(* IEC 61131-3 sources: AXOpen/src/messaging/ctrl/src/IxMessaging, 8 files *)

(* ---- eIxMessageCondition.st ---- *)
NAMESPACE ix.framework.core
    TYPE INTERNAL
        eIxMessageCondition : INT
        (
            Unconditional := 0,
            Active := 10,
            Inactive := 20
        );
    END_TYPE
END_NAMESPACE

(* ---- eIxMessageDigestMethod.st ---- *)
NAMESPACE ix.framework.core
    /// <summary>
    /// Message digest methods used to create fingerprint of a message.
    /// </summary>
    TYPE eIxMessageDigestMethod : INT
    (
        /// <summary>
        /// Fastest method with highest probability of colisions.
        /// </summary>
        CRC8 := 8,

        /// <summary>
        /// Moderate speed method with lower probability of colisions.
        /// </summary>
        CRC16 := 16,

        /// <summary>
        /// Slowest speed method with relatively low probability of colisions.
        /// </summary>
        CRC32 := 32,

        /// <summary>
        /// Messages are not digested the repeated messages won't be filtered out.
        /// Use this option on low performance devices.
        /// </summary>
        NONE := 32767
    );
    END_TYPE
END_NAMESPACE

(* ---- IxConstants.st ---- *)
NAMESPACE ix.framework.core
    TYPE PUBLIC
        IxIntConstants : INT
        (
            MAX_MESSAGE_TEXT_LENGHT := 160,
			MDS_MAX_INDEX := 10
        );
    END_TYPE
END_NAMESPACE

(* ---- IxMessage.st ---- *)
NAMESPACE ix.framework.messaging
    ///<summary>
    /// Complete message details including time stamp, message text, message category, identity of the message provider, context cycle in which the message was posted.
    ///</summary>
    TYPE IxMessage:
        STRUCT
            /// <summary>
            /// Time when the message was posted.
            /// </summary>
            {#ix-attr:[ReadOnly()]}
            TimeStamp : LDATE_AND_TIME;

            /// <summary>
            /// Text of the message.
            /// </summary>
            {#ix-attr:[ReadOnly()]}
            Text : STRING[IxIntConstants#MAX_MESSAGE_TEXT_LENGHT];

            /// <summary>
            /// Identity of the TcoObject that posted this message.
            /// </summary>
            {#ix-attr:[ReadOnly()]}
            Identity : ULINT;

            /// <summary>
            /// Message category of this message. See <see cref="TcoCore.eMessageCategory"/> for detailed informations.
            /// </summary>
            Category : eIxMessageCategory;

            /// <summary>
            /// Context cycle in which the message was posted.
            /// </summary>
            {#ix-attr:[ReadOnly()]}
            Cycle : ULINT;

            /// <summary>
            /// Count of messages of the object in the current cycle.
            /// </summary>
            {#ix-attr:[ReadOnly()]}
            PerCycleCount : USINT;

            /// <summary>
            /// Indicates that the message is expected to be dequeed from the buffer.
            /// </summary>
            ExpectDequeing : BOOL;

            /// <summary>
            /// Indicates that the message must be persisted in the alarm view until acknowledged.
            /// </summary>
            Pinned : BOOL;

            /// <summary>
            /// Stores message digest of this message text.
            /// </summary>
            MessageDigest : DWORD;

            // /// <summary>
            // /// Indicates that the message is active.
            // /// </summary>
            // IsActive : BOOL;
        END_STRUCT;
    END_TYPE
 END_NAMESPACE

(* ---- IxMessageDigest.st ---- *)
NAMESPACE ix.framework.messaging
    CLASS PUBLIC IxMessageDigest
        VAR PUBLIC
            Digest : DWORD;
            Cycle : ULINT;
            Count : ULINT;
            Category : eIxMessageCategory;
        END_VAR
    END_CLASS
END_NAMESPACE

(* ---- IxMessenger.st ---- *)
USING ix.framework.core;
USING System.Strings;
USING System.DateTime;
USING ix.framework.utils;
USING ix.framework.core;
USING ix.framework.messaging;

NAMESPACE ix.framework.messaging
	/// <summary>
	/// Provides mechanism for delivering static messages to the supervising applications (SCADA/HMI).
	/// 	<remarks>
	/// 		<note type="important">
	/// 			Each messenger has a single placeholder for the message; it stores the most important message from the last context cycle.
	/// 			If there are more messages in a single cycle for the same messenger then less important messages are discarded and replaced by
	/// 			the message with the category of higher severity.
	/// 		</note>
	/// 		<note type="important">
	/// 			Messenger can send the data to context logger. There is a maximum limit of 10 different messages per messenger in 2 consecutive context cycles.
	/// 			The messages that exceed this limit won't be logged when `OnEventRisen` logging is set.
	/// 		    Take this behaviour into account when designing your system.
	/// 		</note>
	/// 	</remarks>
	/// </summary>
    CLASS IxMessenger (*EXTENDS IxObject*) IMPLEMENTS IIxMessenger, IIxMessageProperties, IIxMessageTextBuilder, IIxMessageCategorize, IIxMessages
		VAR
			/// <summary>
			/// 	Most important message of this instance of messenger; stores the most important message from the last context cycle.
			/// 	If there are more messages in a single cycle for the same
			/// 	messenger then less important messages are discarded and replaced by the message with the category of higher severity.
			/// </summary>
			_mime : IxMessage;
			_Parent : IIxObject;
            {#ix-attr:[ReadOnly()]}
			_contextIdentity : ULINT;
			{#ix-attr:[CompilerOmits()]}
			_mds : ARRAY[0..IxIntConstants#MDS_MAX_INDEX] OF IxMessageDigest;
			{#ix-attr:[CompilerOmits()]}
			_condition : eIxMessageCondition;
			{#ix-attr:[CompilerOmits()]}
			_pinnable : BOOL;
		END_VAR

		VAR
			{#ix-attr:[CompilerOmits()]}
			tmpMessageText : STRING[IxIntConstants#MAX_MESSAGE_TEXT_LENGHT];
			{#ix-attr:[CompilerOmits()]}
			refStringBuilder : REF_TO StringBuilder;
		END_VAR
		VAR
			{#ix-attr:[CompilerOmits()]}
			_conflictingStringBuilder : StringBuilder;
		END_VAR

		/// <summary>
		/// Gets the Most Important Message of this messenger.
		/// </summary>
		METHOD PUBLIC GetMime : IxMessage
			GetMime := THIS._mime;
		END_METHOD

		/// <summary>
		/// Categorizes and creates the message as 'debug'.
		/// </summary>
		METHOD PUBLIC AsDebug : IIxMessageProperties
			AsDebug := THIS.Post(THIS.StringBuilder()^.AsString(), eIxMessageCategory#Debug);
		END_METHOD

		/// <summary>
		/// Categorizes and creates the message as 'error'.
		/// </summary>
		METHOD PUBLIC AsError : IIxMessageProperties
			AsError := THIS.Post(THIS.StringBuilder()^.AsString(), eIxMessageCategory#Error);
		END_METHOD

		/// <summary>
		/// Categorizes and creates the message as 'fatal'.
		/// </summary>
		METHOD PUBLIC AsFatal : IIxMessageProperties
			AsFatal := THIS.Post(THIS.StringBuilder()^.AsString(), eIxMessageCategory#Fatal);
		END_METHOD

		/// <summary>
		/// Categorizes and creates the message as 'information'.
		/// </summary>
		METHOD PUBLIC AsInfo : IIxMessageProperties
			AsInfo := THIS.Post(THIS.StringBuilder()^.AsString(), eIxMessageCategory#Info);
		END_METHOD

		/// <summary>
		/// Categorizes and creates the message as 'trace'.
		/// </summary>
		METHOD PUBLIC AsTrace : IIxMessageProperties
			AsTrace := THIS.Post(THIS.StringBuilder()^.AsString(), eIxMessageCategory#Trace);
		END_METHOD

		/// <summary>
		/// Categorizes and creates the message as 'warning'.
		/// </summary>
		METHOD PUBLIC AsWarning : IIxMessageProperties
			AsWarning := THIS.Post(THIS.StringBuilder()^.AsString(), eIxMessageCategory#Warning);
		END_METHOD

		/// <summary>
		/// Adds message of 'catastrophic' category to the message queue.
		/// Use this category when there is a situation when the device cannot continue operations due to irrecoverable failure.
		/// </summary>
		METHOD PUBLIC Catastrophic : IIxMessageProperties
			VAR_INPUT
				/// <summary>
				/// Arbitrary message string.
				/// </summary>
				Message : STRING[IxIntConstants#MAX_MESSAGE_TEXT_LENGHT];
			END_VAR
			Catastrophic := THIS.Post(Message, eIxMessageCategory#Catastrophic);
		END_METHOD

		/// <summary>
		/// Adds message of 'critical' category to the message queue.
		/// Use this category when a critical error occured, that is not recoverable by the means of software (reset/restore) and a detailed inspection is required.
		/// </summary>
		METHOD PUBLIC Critical : IIxMessageProperties
			VAR_INPUT
				/// <summary>
				/// Arbitrary message string.
				/// </summary>
				Message : STRING[IxIntConstants#MAX_MESSAGE_TEXT_LENGHT];
			END_VAR
			Critical := THIS.Post(Message, eIxMessageCategory#Critical);
		END_METHOD

		/// <summary>
		/// Adds message of 'debug' category to the message queue.
		/// Use when you need to report debug information for you as programmer.
		/// </summary>
		METHOD PUBLIC Debug : IIxMessageProperties
			VAR_INPUT
				/// <summary>
				/// Arbitrary message string.
				/// </summary>
				Message : STRING[IxIntConstants#MAX_MESSAGE_TEXT_LENGHT];
			END_VAR
			Debug := THIS.Post(Message, eIxMessageCategory#Debug);
		END_METHOD

		/// <summary>
		/// Adds message of 'error' category to the message queue.
		/// Use this categoty when there is a failure that cannot be immediately recovered and an intervention is needed. This is typically a situation when a device fails
		/// to deliver expected result.
		/// Do not use this category to report information about failed process like measurement or detection.
		/// </summary>
		METHOD PUBLIC Error : IIxMessageProperties
			VAR_INPUT
				/// <summary>
				/// Arbitrary message string.
				/// </summary>
				Message : STRING[IxIntConstants#MAX_MESSAGE_TEXT_LENGHT];
			END_VAR
			Error := THIS.Post(Message, eIxMessageCategory#Error);
		END_METHOD

		/// <summary>
		/// Adds message of 'information' category to the message queue.
		/// Use when you want to deliver information to the user, that has only informative character and does not adversely affect a process.
		/// </summary>
		METHOD PUBLIC Info : IIxMessageProperties
			VAR_INPUT
				/// <summary>
				/// Arbitrary message string.
				/// </summary>
				Message : STRING[IxIntConstants#MAX_MESSAGE_TEXT_LENGHT];
			END_VAR
			Info := THIS.Post(Message, eIxMessageCategory#Info);
		END_METHOD

		/// <summary>
		/// Adds message of 'notification' category to the message queue.
		/// Use this category when you want to report a notification that may be of interest to the user, but does not adveresly affect a process.
		/// </summary>
		METHOD PUBLIC Notify : IIxMessageProperties
			VAR_INPUT
				/// <summary>
				/// Arbitrary message string.
				/// </summary>
				Message : STRING[IxIntConstants#MAX_MESSAGE_TEXT_LENGHT];
			END_VAR
			Notify := THIS.Post(Message, eIxMessageCategory#Notification);
		END_METHOD

		/// <summary>
		/// Adds message of 'programming error' category to the message queue.
		/// Use this category to inform about a possible programming error, defect in settings or missing information at a level of programming or system or process settings.
		/// </summary>
		METHOD PUBLIC Programming : IIxMessageProperties
			VAR_INPUT
				/// <summary>
				/// Arbitrary message string.
				/// </summary>
				Message : STRING[IxIntConstants#MAX_MESSAGE_TEXT_LENGHT];
			END_VAR
			Programming := THIS.Post(Message, eIxMessageCategory#ProgrammingError);
		END_METHOD

		/// <summary>
		/// Adds message of 'trace' category to the message queue.
		/// Use when you need to track detailed information about internal states of the program for detailed visibility.
		/// This is lowest level of category that can be used in production, for detailed observation of PLC program.
		/// </summary>
		METHOD PUBLIC Trace : IIxMessageProperties
			VAR_INPUT
				/// <summary>
				/// Arbitrary message string.
				/// </summary>
				Message : STRING[IxIntConstants#MAX_MESSAGE_TEXT_LENGHT];
			END_VAR
			Trace := THIS.Post(Message, eIxMessageCategory#Trace);
		END_METHOD

		/// <summary>
		/// Adds message of 'warning' category to the message queue.
		/// Use this category when you want to report to the user an information about a possible problem, that may adversly affect a process.
		/// Information in this cateogory aims to help the user to identify a problem, the cause of such problem does not necessarily stops the process.
		/// </summary>
		METHOD PUBLIC Warning : IIxMessageProperties
			VAR_INPUT
				/// <summary>
				/// Arbitrary message string.
				/// </summary>
				Message : STRING[IxIntConstants#MAX_MESSAGE_TEXT_LENGHT];
			END_VAR
			Warning := THIS.Post(Message, eIxMessageCategory#Warning);
		END_METHOD

		/// <summary>
		/// Appends string to the message text.
		/// </summary>
		/// <remarks>
		/// <note type="warning">
		/// The size of the resulting string should not be more than '160' characters. The characters exceeding this size will be truncated.
		/// </note>
		/// </remarks>
		METHOD PUBLIC Append : IIxMessageTextBuilder
			VAR_INPUT
				Data : BOOL;
			END_VAR
			THIS.StringBuilder()^.Append(Data);
			Append := THIS;
		END_METHOD

		METHOD PUBLIC Append : IIxMessageTextBuilder
			VAR_INPUT
				Data : BYTE;
			END_VAR
			THIS.StringBuilder()^.Append(Data);
			Append := THIS;
		END_METHOD

		METHOD PUBLIC Append : IIxMessageTextBuilder
			VAR_INPUT
				Data : WORD;
			END_VAR
			THIS.StringBuilder()^.Append(Data);
			Append := THIS;
		END_METHOD

		METHOD PUBLIC Append : IIxMessageTextBuilder
			VAR_INPUT
				Data : DWORD;
			END_VAR
			THIS.StringBuilder()^.Append(Data);
			Append := THIS;
		END_METHOD

		METHOD PUBLIC Append : IIxMessageTextBuilder
			VAR_INPUT
				Data : LWORD;
			END_VAR
			THIS.StringBuilder()^.Append(Data);
			Append := THIS;
		END_METHOD

		METHOD PUBLIC Append : IIxMessageTextBuilder
			VAR_INPUT
				Data : SINT;
			END_VAR
			THIS.StringBuilder()^.Append(Data);
			Append := THIS;
		END_METHOD

		METHOD PUBLIC Append : IIxMessageTextBuilder
			VAR_INPUT
				Data : INT;
			END_VAR
			THIS.StringBuilder()^.Append(Data);
			Append := THIS;
		END_METHOD

		METHOD PUBLIC Append : IIxMessageTextBuilder
			VAR_INPUT
				Data : DINT;
			END_VAR
			THIS.StringBuilder()^.Append(Data);
			Append := THIS;
		END_METHOD

		METHOD PUBLIC Append : IIxMessageTextBuilder
			VAR_INPUT
				Data : LINT;
			END_VAR
			THIS.StringBuilder()^.Append(Data);
			Append := THIS;
		END_METHOD

		METHOD PUBLIC Append : IIxMessageTextBuilder
			VAR_INPUT
				Data : USINT;
			END_VAR
			THIS.StringBuilder()^.Append(Data);
			Append := THIS;
		END_METHOD

		METHOD PUBLIC Append : IIxMessageTextBuilder
			VAR_INPUT
				Data : UINT;
			END_VAR
			THIS.StringBuilder()^.Append(Data);
			Append := THIS;
		END_METHOD

		METHOD PUBLIC Append : IIxMessageTextBuilder
			VAR_INPUT
				Data : UDINT;
			END_VAR
			THIS.StringBuilder()^.Append(Data);
			Append := THIS;
		END_METHOD

		METHOD PUBLIC Append : IIxMessageTextBuilder
			VAR_INPUT
				Data : ULINT;
			END_VAR
			THIS.StringBuilder()^.Append(Data);
			Append := THIS;
		END_METHOD

		METHOD PUBLIC Append : IIxMessageTextBuilder
			VAR_INPUT
				Data : REAL;
			END_VAR
			THIS.StringBuilder()^.Append(Data);
			Append := THIS;
		END_METHOD

		METHOD PUBLIC Append : IIxMessageTextBuilder
			VAR_INPUT
				Data : LREAL;
			END_VAR
			THIS.StringBuilder()^.Append(Data);
			Append := THIS;
		END_METHOD

		METHOD PUBLIC Append : IIxMessageTextBuilder
			VAR_INPUT
				Data : TIME;
			END_VAR
			THIS.StringBuilder()^.Append(Data);
			Append := THIS;
		END_METHOD

		METHOD PUBLIC Append : IIxMessageTextBuilder
			VAR_INPUT
				Data : LTIME;
			END_VAR
			THIS.StringBuilder()^.Append(Data);
			Append := THIS;
		END_METHOD

		METHOD PUBLIC Append : IIxMessageTextBuilder
			VAR_INPUT
				Data : DATE;
			END_VAR
			THIS.StringBuilder()^.Append(Data);
			Append := THIS;
		END_METHOD

		METHOD PUBLIC Append : IIxMessageTextBuilder
			VAR_INPUT
				Data : LDATE;
			END_VAR
			THIS.StringBuilder()^.Append(Data);
			Append := THIS;
		END_METHOD

		METHOD PUBLIC Append : IIxMessageTextBuilder
			VAR_INPUT
				Data : TIME_OF_DAY;
			END_VAR
			THIS.StringBuilder()^.Append(Data);
			Append := THIS;
		END_METHOD

		METHOD PUBLIC Append : IIxMessageTextBuilder
			VAR_INPUT
				Data : LTIME_OF_DAY;
			END_VAR
			THIS.StringBuilder()^.Append(Data);
			Append := THIS;
		END_METHOD

		METHOD PUBLIC Append : IIxMessageTextBuilder
			VAR_INPUT
				Data : DATE_AND_TIME;
			END_VAR
			THIS.StringBuilder()^.Append(Data);
			Append := THIS;
		END_METHOD

		METHOD PUBLIC Append : IIxMessageTextBuilder
			VAR_INPUT
				Data : LDATE_AND_TIME;
			END_VAR
			THIS.StringBuilder()^.Append(Data);
			Append := THIS;
		END_METHOD

		METHOD PUBLIC Append : IIxMessageTextBuilder
			VAR_INPUT
				Data : CHAR;
			END_VAR
			THIS.StringBuilder()^.Append(Data);
			Append := THIS;
		END_METHOD

		// METHOD PUBLIC Append : IIxMessageTextBuilder
		// 	VAR_INPUT
		// 		Data : WCHAR;
		// 	END_VAR
		// 	THIS.StringBuilder()^.Append(Data);
		// 	Append := THIS;
		// END_METHOD

		METHOD PUBLIC Append : IIxMessageTextBuilder
			VAR_INPUT
				Data : STRING[IxIntConstants#MAX_MESSAGE_TEXT_LENGHT];
			END_VAR
			THIS.StringBuilder()^.Append(Data);
			Append := THIS;
		END_METHOD

		// METHOD PUBLIC Append : IIxMessageTextBuilder
		// 	VAR_INPUT
		// 		Data : WSTRING[IxIntConstants#MAX_MESSAGE_TEXT_LENGHT];
		// 	END_VAR
		// 	THIS.StringBuilder()^.Append(Data);
		// 	Append := THIS;
		// END_METHOD

		/// <summary>
		/// Gets categorization methods for fluent message builder.
		/// </summary>
		METHOD PUBLIC As : IIxMessageCategorize
			As := THIS;
		END_METHOD

		/// <summary>
		/// Initiates new message text building for this messenger in fluent-like fashion.
		/// </summary>
		METHOD PUBLIC Build : IIxMessageTextBuilder
			THIS.StringBuilder()^.Clear();
			Build := THIS;
		END_METHOD

		/// <summary>
		/// Clears the message content.
		/// </summary>
		METHOD PUBLIC Clear
			NewDateAndTime(1970, 1, 1, 0, 0, 0, 0, 0, 0, _mime.TimeStamp);
			_mime.Text := '';
			_mime.Identity := ULINT#0;
			_mime.Category := eIxMessageCategory#All;
			_mime.Cycle := ULINT#0;
			_mime.PerCycleCount := USINT#0;
			_mime.Pinned := FALSE;
		END_METHOD

		METHOD PROTECTED Compose : IxMessage
			VAR_INPUT
				/// <summary>
				/// Arbitrary message string.
				/// </summary>
				Message : STRING[IxIntConstants#MAX_MESSAGE_TEXT_LENGHT];
				/// <summary>
				/// Message category.
				/// </summary>
				Category : eIxMessageCategory;
			END_VAR
					Compose.TimeStamp :=  _Parent.GetContext().GetRtc().NowUTC();
					Compose.Text := Message;
					Compose.Identity := _Parent.GetIdentity();
					Compose.Category := Category;
					Compose.Cycle := _Parent.GetContext().OpenCycleCount();
					// Compose.MessageDigest := THIS.Digest(Message, _Parent.GetContext().Environment().Messaging().GetMessageDigestMethod());
					Compose.MessageDigest := THIS.Digest(Message,eIxMessageDigestMethod#CRC32);
		END_METHOD

		METHOD PRIVATE Digest: DWORD
			VAR_INPUT
				Message : STRING[254];
				inDigestType : eIxMessageDigestMethod;
			END_VAR

			CASE inDigestType OF
				eIxMessageDigestMethod#CRC8 :
					Digest := IxCRC_8(Message);
					eIxMessageDigestMethod#CRC16 :
					Digest := IxCRC_16(Message);
					eIxMessageDigestMethod#CRC32 :
					Digest := IxCRC_32(Message);
				ELSE
					Digest := DWORD#0;
			END_CASE;
		END_METHOD

		METHOD PUBLIC Initialize
			VAR_INPUT
				ParentObject : IIxObject;
			END_VAR
			_Parent := ParentObject;
			_contextIdentity := ParentObject.GetIdentity();
		END_METHOD

		METHOD PUBLIC OnCondition : IIxMessages
			VAR_INPUT
				inCondition : BOOL;
			END_VAR
			IF (inCondition) THEN
				_condition := eIxMessageCondition#Active;
			ELSE
				_condition := eIxMessageCondition#Inactive;
			END_IF;

			OnCondition := THIS;
		END_METHOD

		/// <summary>
		/// 	Pins this message that no other message will override it.
		/// 	The messenger won't accept new messages until acknowledged in diagnostics view by user, unipenned by `Unpin()` methods or cleared by `Clear()` method
		/// 	of this messenger.
		/// </summary>
		/// <note type="important">
		/// 	Pinned messages do no accept incomming messages on the same messenger. The incomming messages will be though the context logger when active.
		/// </note>
		METHOD PUBLIC Pin: IIxMessageProperties
			IF NOT(_Parent = NULL) THEN
				IF NOT(_Parent.GetContext()= NULL) THEN
					IF(_pinnable) THEN
						IF(_mime.Cycle = _Parent.GetContext().OpenCycleCount())THEN
							_mime.Pinned := TRUE;
						END_IF;
					END_IF;
				END_IF;
			END_IF;
			Pin := THIS;
		END_METHOD

		/// <summary>
		/// Gets `true` when this messenger is pinned (awaiting acknowledgement in diagnostics view).
		/// </summary>
		METHOD PUBLIC IsPinned: BOOL
			IsPinned := FALSE;
			IF _mime.Pinned THEN
				IsPinned :=  tmpMessageText = _mime.Text;
			END_IF;
		END_METHOD

		/// <summary>
		/// Gets `true` when this messenger is active.
		/// </summary>
		METHOD PUBLIC IsActive: BOOL
			IsActive := _mime.Cycle = _Parent.GetContext().OpenCycleCount() OR _mime.Pinned ;
		END_METHOD

		/// <summary>
		/// Creates message of given category for this messenger.
		/// </summary>
		METHOD PUBLIC Post : IIxMessageProperties
			VAR_INPUT
				/// <summary>
				/// Arbitrary message string.
				/// </summary>
				Message : STRING[IxIntConstants#MAX_MESSAGE_TEXT_LENGHT];
				/// <summary>
				/// Message category.
				/// </summary>
				Category : eIxMessageCategory;
			END_VAR

			VAR
				_wouldBeMime : IxMessage;
			END_VAR

			Post := THIS;

			tmpMessageText := Message;

			_pinnable := FALSE;

			IF(_condition = eIxMessageCondition#Inactive) THEN
				_condition := eIxMessageCondition#Unconditional;
				RETURN;
			END_IF;

			_condition := eIxMessageCondition#Unconditional;

							IF(Category < _Parent.GetContext().Environment().Messaging().GetMinLevel()
								OR _Parent.GetContext().Environment().Messaging().IsSuspended()) THEN
									RETURN;
							END_IF;

							IF (NOT _mime.Pinned) THEN
								_mime.PerCycleCount := _mime.PerCycleCount + USINT#1;
								_wouldBeMime := THIS.Compose(Message, Category);
								_wouldBeMime.PerCycleCount := _mime.PerCycleCount;
							ELSIF _mime.Pinned THEN
								IF(_mime.Text <>  Message OR _mime.Category <> Category) THEN
									IF(	_mime.PerCycleCount < 255) THEN
										_mime.PerCycleCount := _mime.PerCycleCount + USINT#1;
									END_IF;
								END_IF;
							END_IF;

							// Same cycle filter for most important messge.
							IF(_mime.Cycle = _Parent.GetContext().OpenCycleCount()) THEN
								IF(_wouldBeMime.Category > _mime.Category)
								AND (NOT _mime.Pinned) THEN
									_mime := _wouldBeMime;
								END_IF;
							ELSE
							// Different cycle
								IF (NOT _mime.Pinned) THEN
									_wouldBeMime.PerCycleCount := USINT#1;
									_mime := _wouldBeMime;
								END_IF;
							END_IF;

							_pinnable := TRUE;
		END_METHOD

		METHOD PUBLIC StringBuilder : REF_TO StringBuilder
			IF(NOT(refStringBuilder = NULL)) THEN
				StringBuilder := refStringBuilder;
			ELSE
				StringBuilder := REF(_conflictingStringBuilder);
			END_IF;
		END_METHOD

		METHOD PUBLIC UnPin
			_mime.Pinned := FALSE;
		END_METHOD
	END_CLASS
END_NAMESPACE

(* ---- IxMessengerEnv.st ---- *)
USING ix.framework.utils;
using ix.framework.core;

NAMESPACE ix.framework.messaging
    CLASS PUBLIC IxMessengerEnv IMPLEMENTS IIxMessengerEnv
		VAR
			_minLevel : eIxMessageCategory;
			_isMessagingSuspended : BOOL;
			_messageDigestMethod : eIxMessageDigestMethod := eIxMessageDigestMethod#CRC16;
			//_messengerLoggingMethod : eIxMessengerLogMethod := eIxMessengerLogMethod#OnEventRisen;
			_sb : REF_TO StringBuilder;
		END_VAR

		/// <inheritdoc />
		METHOD PUBLIC IsSuspended: BOOL
			IsSuspended := _isMessagingSuspended;
		END_METHOD

		/// <inheritdoc />
		METHOD PUBLIC GetMessageDigestMethod : eIxMessageDigestMethod
			GetMessageDigestMethod := _messageDigestMethod;
		END_METHOD

		/// <inheritdoc />
		METHOD PUBLIC SetMessageDigestMethod
			VAR_INPUT
				inDigestMethod : eIxMessageDigestMethod;
			END_VAR
			_messageDigestMethod := inDigestMethod;
		END_METHOD

		/// <inheritdoc />
		METHOD PUBLIC GetMinLevel : eIxMessageCategory
			GetMinLevel := _minLevel;
		END_METHOD

		/// <inheritdoc />
		METHOD PUBLIC SetMinLevel
			VAR_INPUT
				inMessageCategory : eIxMessageCategory;
			END_VAR
			_minLevel := inMessageCategory;
		END_METHOD

		/// <inheritdoc />
		METHOD PUBLIC Resume
			_isMessagingSuspended := FALSE;
		END_METHOD

		/// <inheritdoc />
		METHOD PUBLIC Suspend
			_isMessagingSuspended := TRUE;
		END_METHOD

		/// <inheritdoc />
		METHOD PUBLIC GetStringBuilder : REF_TO StringBuilder
			GetStringBuilder ?= _sb;
		END_METHOD
	END_CLASS
END_NAMESPACE

(* ---- eIxMessageCategory.st ---- *)
NAMESPACE ix.framework.core
    TYPE PUBLIC
        ///<summary>
        /// Message categories.
        /// ATTENTION: Values must be multiply of 100
        ///</summary>
        eIxMessageCategory : INT
        (
            All := 0,

            ///<summary>
            /// Trace message to be used for tracing purpose.
            /// Use when you need to track detailed information about internal states of the program for detailed visibility.
            /// This is lowest level of category that can be used in production, for detailed observation of PLC program.
            ///</summary>
            Trace := 100,

            ///<summary>
            /// Debug message to be used for debugging purpose only.
            /// Use when you need to report debug information for you as programmer.
            ///</summary>
            Debug := 200,

            ///<summary>
            /// Info message.
            /// Use when you want to deliver information to the user, that has only informative character and does not adversely affect a process.
            ///</summary>
            Info := 300,

            ///<summary>
            /// Time-out message.
            /// Use this category when you want to report a timed-out information, that may eventually succed.
            ///</summary>
            TimedOut := 400,

            ///<summary>
            /// Notification message.
            /// Use this category when you want to report a notification that may be of interest to the user, but does not adversly affect a process.
            ///</summary>
            Notification := 500,

            ///<summary>
            /// Warning message.
            /// Use this category when you want to report to the user an information about a possible problem, that may adversly affect a process.
            /// Information in this cateogory aims to help the user to identify a problem, the cause of such problem does not necessarily stops the process.
            ///</summary>
            Warning := 600,

            ///<summary>
            /// Error message.
            /// Use this categoty when there is a failure that cannot be immediately recovered and an intervention is needed. This is typically a situation when a device fails
            /// to deliver expected result.
            /// Do not use this category to report information about failed process like measurement or detection.
            ///</summary>
            Error := 700,

            ///<summary>
            /// Programming issue.
            /// Use this category to inform about a possible programming error, defect in settings or missing information at a level of programming or system or process settings.
            ///</summary>
            ProgrammingError := 900,

            ///<summary>
            /// Critical error.
            /// Use this category when a critical error occured, that is not recoverable by the means of software (reset/restore) but device still operates under such conditions; a detailed inspection and an expert action is required.
            ///</summary>
            Critical := 1000,

            ///<summary>
            /// Fatal error.
            /// Use this category when a fatal error occured, that is not recoverable by the means of software (reset/restore) and a detailed inspection is required, the device is not able to continue without special intervention,
            ///</summary>
            Fatal    := 1100,

            ///<summary>
            /// Catastrophic error.
            /// Use this category when there is a situation when the device cannot continue operations due to irrecoverable failure.
            ///</summary>
            Catastrophic := 1200,

            None := 32000
        );
    END_TYPE
END_NAMESPACE
